VAR_INPUT
	input1 : INT;
	input2 : BOOL;
END_VAR
BEGIN
	// Some code here
END_FUNCTION_BLOCK
